(* IEC 61131-3 sources: plc_on_fpga_riscv_hybrid/RV_FPGA_PLC_IDE_Projects/Test_Project, 1 file *)

(* ---- Test_Project.il ---- *)
VAR
    X   : INT
    Y   : INT
    Z   : INT
    TON   : TON_1
END_VAR

PROGRAM Test_Project
    R1 :
        LD     15
        ST     X
    R2 :
        LD     20
        ST     Y
    R3 :
        LD     X
        ADD    Y
        ST     Z
        CAL TON_1(
            IN := %SW.0,
            PT := X,
            ET := Z,
            Q  => %LEDG.0)
END_PROGRAM
